// TIA Portal V20 export
DATA_BLOCK "BK09"   // DB235
// stored: MemoryReserve 100
   VAR
      "X10-1 SIDE TAPE CUTTER BACKWARD" : Bool;
      "X11-1 SIDE TAPE CUTTER CLAMP BACKWARD" : Bool;
      "X12-1 SIDE TAPE CLAMP OPEN" : Bool;
      "X13-1 SIDE TAPE TENSION BACKWARD" : Bool;
      "X14-1 SIDE TAPE LOADING BACKWARD" : Bool;
      "X15-1 SIDE TAPE DIAMETER SENSOR" : Bool;
      "X16-1 SPARE" : Bool;
      "X17-1 SPARE" : Bool;
      "X10-2 SIDE TAPE CUTTER FORWARD" : Bool;
      "X11-2 SIDE TAPE CUTTER CLAMP FORWARD" : Bool;
      "X12-2 SIDE TAPE CLAMP CLOSE" : Bool;
      "X13-2 SIDE TAPE TENSION FORWARD" : Bool;
      "X14-2 SIDE TAPE LOADING FORWARD" : Bool;
      "X15-2 SPARE" : Bool;
      "X16-2 SPARE" : Bool;
      "X17-2 SPARE" : Bool;
   END_VAR
BEGIN
END_DATA_BLOCK
